FUNCTION_BLOCK FB_PlantControl_B57

VAR
	Plant_Control : PlantAndCMs.FB_PlantControl_V2;
	
	
	MB_START : BOOL;
	MB_EMG_STOP : BOOL;
END_VAR

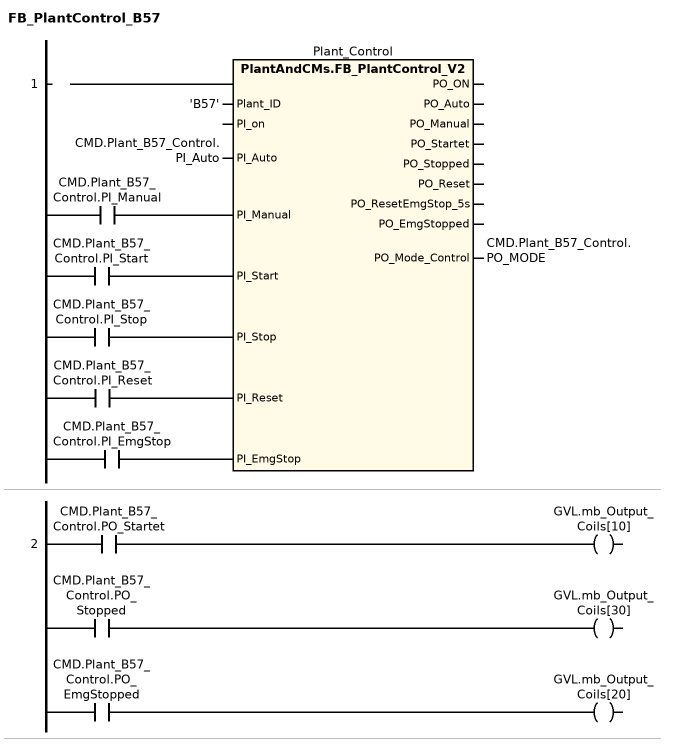
// NETWORK 1
Plant_Control(
    Plant_ID := 'B57',
    PI_Auto := CMD.Plant_B57_Control.PI_Auto,
    PI_Manual := CMD.Plant_B57_Control.PI_Manual,
    PI_Start := CMD.Plant_B57_Control.PI_Start,
    PI_Stop := CMD.Plant_B57_Control.PI_Stop,
    PI_Reset := CMD.Plant_B57_Control.PI_Reset,
    PI_EmgStop := CMD.Plant_B57_Control.PI_EmgStop,
    PO_Mode_Control => CMD.Plant_B57_Control.PO_MODE); // PlantAndCMs.FB_PlantControl_V2

// NETWORK 2
GVL.mb_Output_Coils[10] := CMD.Plant_B57_Control.PO_Startet;
GVL.mb_Output_Coils[30] := CMD.Plant_B57_Control.PO_Stopped;
GVL.mb_Output_Coils[20] := CMD.Plant_B57_Control.PO_EmgStopped;

END_FUNCTION_BLOCK

(* stored: Version 1.1.0.1, ProductVersion 3.1.4024.13
   POU FB_PlantControl_B57: Id {9284e2b2-e942-4516-90ef-e844f5f4e9d8}, SpecialFunc None *)
